{attribute 'qualified_only'}
VAR_GLOBAL
	Inputs AT %I* : ARRAY[0..7] OF BOOL;
	Outputs  AT %Q* : ARRAY[0..7] OF BOOL;
END_VAR

(* stored: Version 1.1.0.1, ProductVersion 3.1.4024.6
   GVL gMANIPULATOR_IO: Id {cb092603-2ff9-4dc2-8c6e-b8358833817b} *)
